Staubli VAL3: RectanglePoint.pgx

public program RectanglePoint(trsf& x_trSource[], trsf& x_trDest[], bool& x_bRes)
  local frame l_fFrame
  local num l_Dia
  local num l_nLegth
  local point l_pBuff
begin
  //矩形

  //根据三个trsf建立frame
  call SetFrame(x_trSource,l_fFrame,x_bRes)
  if !x_bRes
    return
  endIf


  //矩形的宽
  l_Dia=distance(x_trSource[1],x_trSource[2])
  //矩形的长
  l_nLegth=distance(x_trSource[0],x_trSource[1])



  link(l_pBuff,l_fFrame)
  l_pBuff.trsf={l_nLegth/2,0,0,0,0,0}
  x_trDest[0]=position(l_pBuff,world)

  l_pBuff.trsf={l_nLegth,0,0,0,0,0}
  x_trDest[1]=position(l_pBuff,world)

  l_pBuff.trsf={l_nLegth,l_Dia,0,0,0,0}
  x_trDest[2]=position(l_pBuff,world)

  l_pBuff.trsf={0,l_Dia,0,0,0,0}
  x_trDest[3]=position(l_pBuff,world)


  l_pBuff.trsf={0,0,0,0,0,0}
  x_trDest[4]=position(l_pBuff,world)

  x_trDest[5]=x_trDest[0]

    //圆心点
  l_pBuff.trsf={l_nLegth/2,min(l_nLegth/2,l_Dia/2),0,0,0,0}
  x_trDest[20]=position(l_pBuff,world)


end
